PROGRAM Circuito_L12
VAR_INPUT
	Modo_Calibrar_L12: BOOL;
END_VAR
VAR
	fbBomba_L12 :Equipo_Motor_ATV320;
	ControlValv_ioLink_V1:ControlValv_ioLink;
	ControlValv_ioLink_V2: ControlValv_ioLink;
	ControlValv_ioLink_V3: ControlValv_ioLink;
	ControlValv_ioLink_V4: ControlValv_ioLink;
	Falla_L12_V1:BOOL;
	Falla_L12_V2:BOOL;
	Falla_L12_V3:BOOL;
	Falla_L12_V4:BOOL;
	Balanza_PU3_WT12: Balanza;
	dHS:DINT;
	TOF_calibradoIBC: TOF;
	PID_L12_SP:REAL;
	PID_L12_auto:BOOL;
	PID_L12_reset:BOOL;
	PID_L12_manual:REAL;
	PID_L12_bMuerta:REAL := 5;
	PID_L12_Kp:REAL := 0.1;
	PID_L12_Ti:REAL := 100;
	PID_L12_PV:REAL;
	Dosis_L12:REAL;
	TiempoInyeccion_L12	:DINT;
	Peso	:REAL;
	Offset_L12:REAL;
	Inyeccion_L12:BOOL;

	Volumen_L12:REAL;
	Calculo_caudal_L12: Calculo_caudal;
	CorrecionCaudalxOffset_L12: CorrecionCaudalxOffset;
	tInyeccion: TON;
	Total :REAL;
	Totalant	:REAL;
	auxIniCal:BOOL;
	AuxVol12:REAL;
	TDemoraInyectar: TON;
	SetDemoraInyeccion: REAL;
	Tiempo_seg_to_TIME_DemoraInyec: Tiempo_seg_to_TIME;
	AuxTDemoraInyec: TIME;
	PID_L12: FB_PID;
	Tiempo_TIME_to_seg_InyCal: Tiempo_TIME_to_seg;
	AuxInyCal:TIME;
	IniTotalFT2:REAL;
	Auxconsumo:REAL;
	ProductoAsociado: STRING;
	Lavagem_Circuito12: Lavagem;
	Filtro:Filtro2;
	BasicPID_L12: FB_BasicPID;
	TON_StartBomba: TON;
END_VAR

VAR PERSISTENT
	UltimaCalibracao	:UDINT;	//Data e hora da ultima calibração
END_VAR
VAR // added by the converter: edge detectors and wires of the graphical bodies
    _w1, _w2, _w3, _w4, _w5, _w6, _w7, _w8, _w9, _w10, _w11, _w12, _w13 : BOOL;
    _ft1 : F_TRIG;
    _rt1, _rt2, _rt3 : R_TRIG;
END_VAR

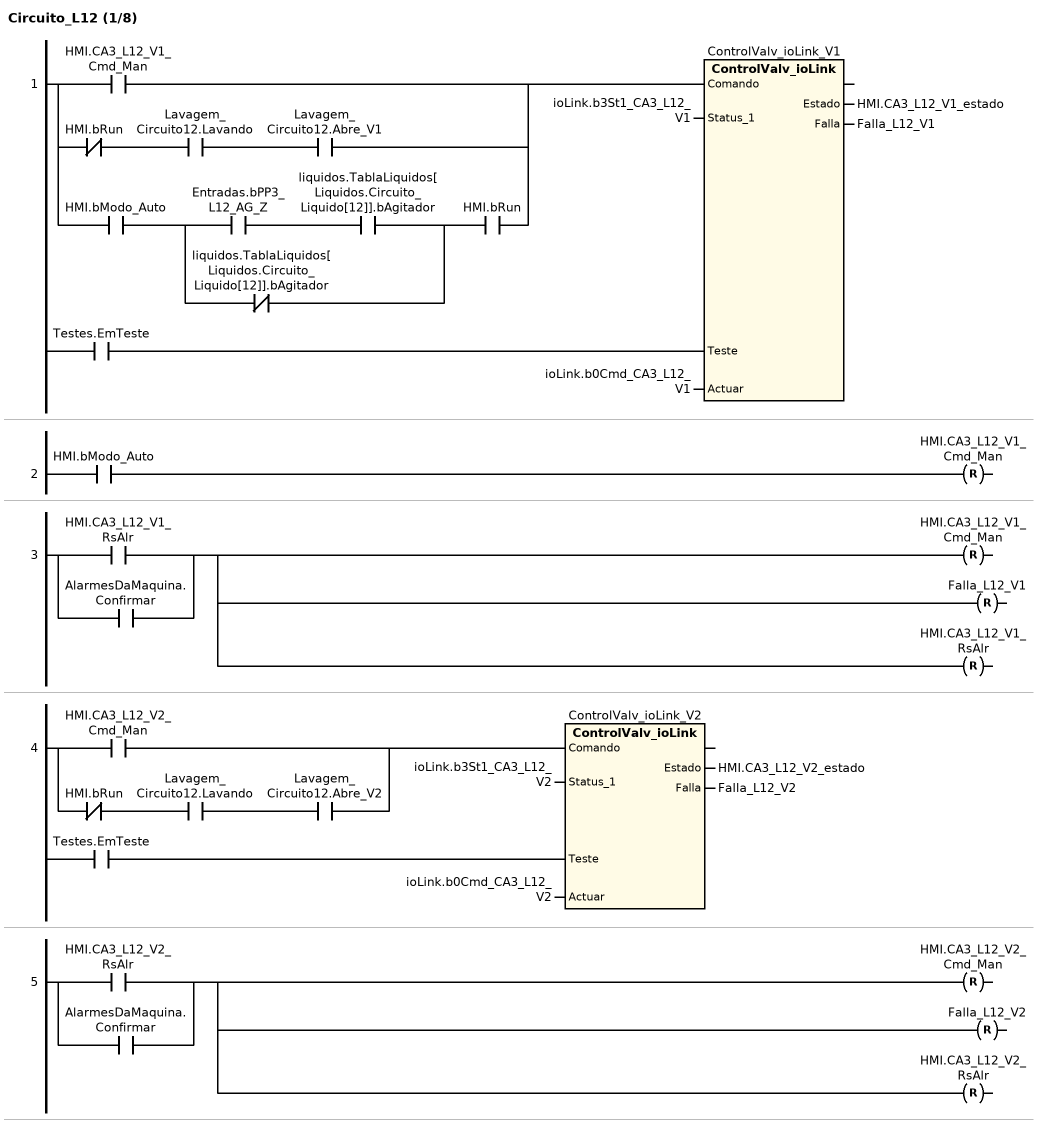
// NETWORK 1
ControlValv_ioLink_V1(
    Comando := HMI.CA3_L12_V1_Cmd_Man OR NOT HMI.bRun AND Lavagem_Circuito12.Lavando AND Lavagem_Circuito12.Abre_V1 OR HMI.bModo_Auto AND (Entradas.bPP3_L12_AG_Z AND (liquidos.TablaLiquidos[Liquidos.Circuito_Liquido[12]].bAgitador) OR NOT (liquidos.TablaLiquidos[Liquidos.Circuito_Liquido[12]].bAgitador)) AND HMI.bRun,
    Status_1 := ioLink.b3St1_CA3_L12_V1,
    Teste := Testes.EmTeste,
    Actuar := ioLink.b0Cmd_CA3_L12_V1,
    Estado => HMI.CA3_L12_V1_estado,
    Falla => Falla_L12_V1); // ControlValv_ioLink

// NETWORK 2
HMI.CA3_L12_V1_Cmd_Man R= HMI.bModo_Auto;

// NETWORK 3
_w1 := HMI.CA3_L12_V1_RsAlr OR AlarmesDaMaquina.Confirmar;
HMI.CA3_L12_V1_Cmd_Man R= _w1;
Falla_L12_V1 R= _w1;
HMI.CA3_L12_V1_RsAlr R= _w1;

// NETWORK 4
ControlValv_ioLink_V2(
    Comando := HMI.CA3_L12_V2_Cmd_Man OR NOT HMI.bRun AND Lavagem_Circuito12.Lavando AND Lavagem_Circuito12.Abre_V2,
    Status_1 := ioLink.b3St1_CA3_L12_V2,
    Teste := Testes.EmTeste,
    Actuar := ioLink.b0Cmd_CA3_L12_V2,
    Estado => HMI.CA3_L12_V2_estado,
    Falla => Falla_L12_V2); // ControlValv_ioLink

// NETWORK 5
_w2 := HMI.CA3_L12_V2_RsAlr OR AlarmesDaMaquina.Confirmar;
HMI.CA3_L12_V2_Cmd_Man R= _w2;
Falla_L12_V2 R= _w2;
HMI.CA3_L12_V2_RsAlr R= _w2;

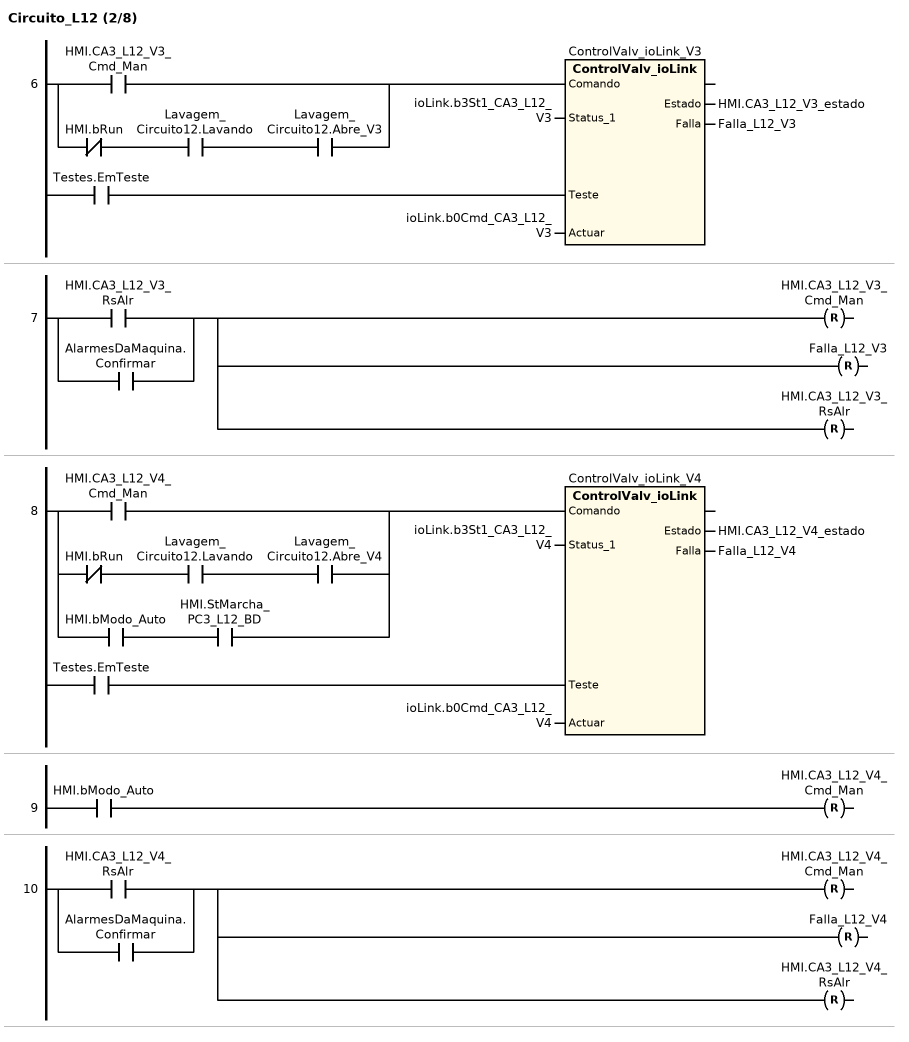
// NETWORK 6
ControlValv_ioLink_V3(
    Comando := HMI.CA3_L12_V3_Cmd_Man OR NOT HMI.bRun AND Lavagem_Circuito12.Lavando AND Lavagem_Circuito12.Abre_V3,
    Status_1 := ioLink.b3St1_CA3_L12_V3,
    Teste := Testes.EmTeste,
    Actuar := ioLink.b0Cmd_CA3_L12_V3,
    Estado => HMI.CA3_L12_V3_estado,
    Falla => Falla_L12_V3); // ControlValv_ioLink

// NETWORK 7
_w3 := HMI.CA3_L12_V3_RsAlr OR AlarmesDaMaquina.Confirmar;
HMI.CA3_L12_V3_Cmd_Man R= _w3;
Falla_L12_V3 R= _w3;
HMI.CA3_L12_V3_RsAlr R= _w3;

// NETWORK 8
ControlValv_ioLink_V4(
    Comando := HMI.CA3_L12_V4_Cmd_Man OR NOT HMI.bRun AND Lavagem_Circuito12.Lavando AND Lavagem_Circuito12.Abre_V4 OR HMI.bModo_Auto AND HMI.StMarcha_PC3_L12_BD,
    Status_1 := ioLink.b3St1_CA3_L12_V4,
    Teste := Testes.EmTeste,
    Actuar := ioLink.b0Cmd_CA3_L12_V4,
    Estado => HMI.CA3_L12_V4_estado,
    Falla => Falla_L12_V4); // ControlValv_ioLink

// NETWORK 9
HMI.CA3_L12_V4_Cmd_Man R= HMI.bModo_Auto;

// NETWORK 10
_w4 := HMI.CA3_L12_V4_RsAlr OR AlarmesDaMaquina.Confirmar;
HMI.CA3_L12_V4_Cmd_Man R= _w4;
Falla_L12_V4 R= _w4;
HMI.CA3_L12_V4_RsAlr R= _w4;

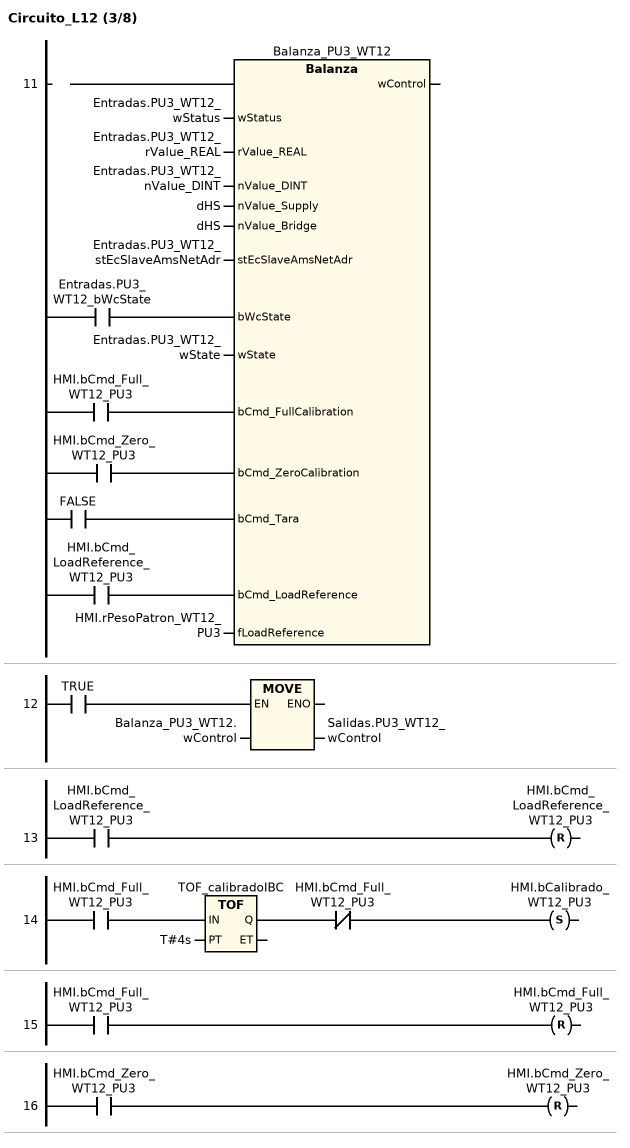
// NETWORK 11
Balanza_PU3_WT12(
    wStatus := Entradas.PU3_WT12_wStatus,
    rValue_REAL := Entradas.PU3_WT12_rValue_REAL,
    nValue_DINT := Entradas.PU3_WT12_nValue_DINT,
    nValue_Supply := dHS,
    nValue_Bridge := dHS,
    stEcSlaveAmsNetAdr := Entradas.PU3_WT12_stEcSlaveAmsNetAdr,
    bWcState := Entradas.PU3_WT12_bWcState,
    wState := Entradas.PU3_WT12_wState,
    bCmd_FullCalibration := HMI.bCmd_Full_WT12_PU3,
    bCmd_ZeroCalibration := HMI.bCmd_Zero_WT12_PU3,
    bCmd_Tara := FALSE,
    bCmd_LoadReference := HMI.bCmd_LoadReference_WT12_PU3,
    fLoadReference := HMI.rPesoPatron_WT12_PU3); // Balanza

// NETWORK 12
Salidas.PU3_WT12_wControl := Balanza_PU3_WT12.wControl;

// NETWORK 13
HMI.bCmd_LoadReference_WT12_PU3 R= HMI.bCmd_LoadReference_WT12_PU3;

// NETWORK 14
TOF_calibradoIBC(IN := HMI.bCmd_Full_WT12_PU3, PT := T#4s); // TOF
HMI.bCalibrado_WT12_PU3 S= TOF_calibradoIBC.Q AND NOT HMI.bCmd_Full_WT12_PU3;

// NETWORK 15
HMI.bCmd_Full_WT12_PU3 R= HMI.bCmd_Full_WT12_PU3;

// NETWORK 16
HMI.bCmd_Zero_WT12_PU3 R= HMI.bCmd_Zero_WT12_PU3;

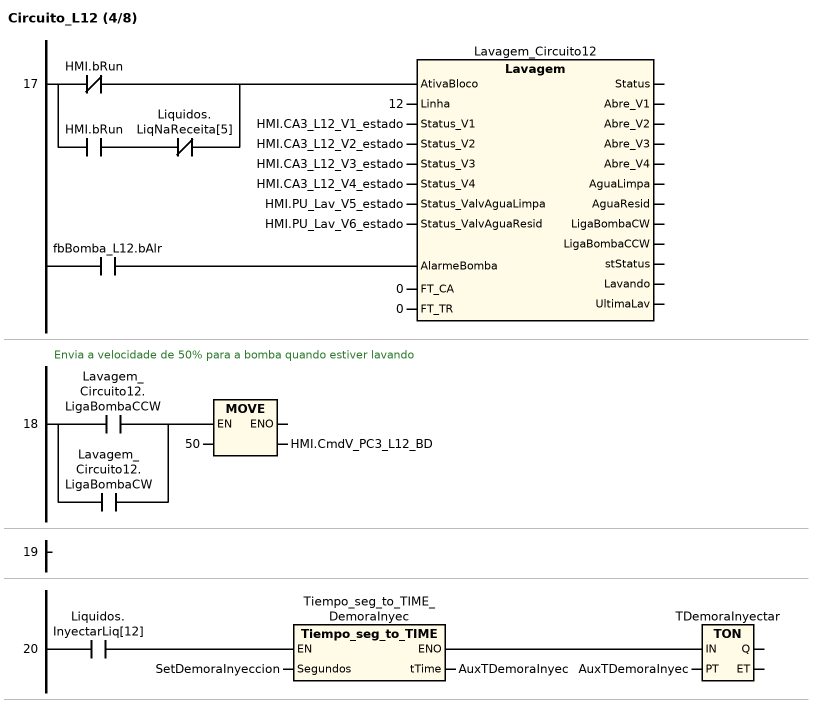
// NETWORK 17
Lavagem_Circuito12(
    AtivaBloco := NOT HMI.bRun OR HMI.bRun AND NOT Liquidos.LiqNaReceita[5],
    Linha := 12,
    Status_V1 := HMI.CA3_L12_V1_estado,
    Status_V2 := HMI.CA3_L12_V2_estado,
    Status_V3 := HMI.CA3_L12_V3_estado,
    Status_V4 := HMI.CA3_L12_V4_estado,
    Status_ValvAguaLimpa := HMI.PU_Lav_V5_estado,
    Status_ValvAguaResid := HMI.PU_Lav_V6_estado,
    AlarmeBomba := fbBomba_L12.bAlr,
    FT_CA := 0,
    FT_TR := 0); // Lavagem

// NETWORK 18
// Envia a velocidade de 50% para a bomba quando estiver lavando
IF Lavagem_Circuito12.LigaBombaCCW OR Lavagem_Circuito12.LigaBombaCW THEN HMI.CmdV_PC3_L12_BD := 50; END_IF

// NETWORK 19

// NETWORK 20
_w5 := Liquidos.InyectarLiq[12];
IF _w5 THEN
    Tiempo_seg_to_TIME_DemoraInyec(Segundos := SetDemoraInyeccion, tTime => AuxTDemoraInyec); // Tiempo_seg_to_TIME
END_IF
TDemoraInyectar(IN := _w5, PT := AuxTDemoraInyec); // TON

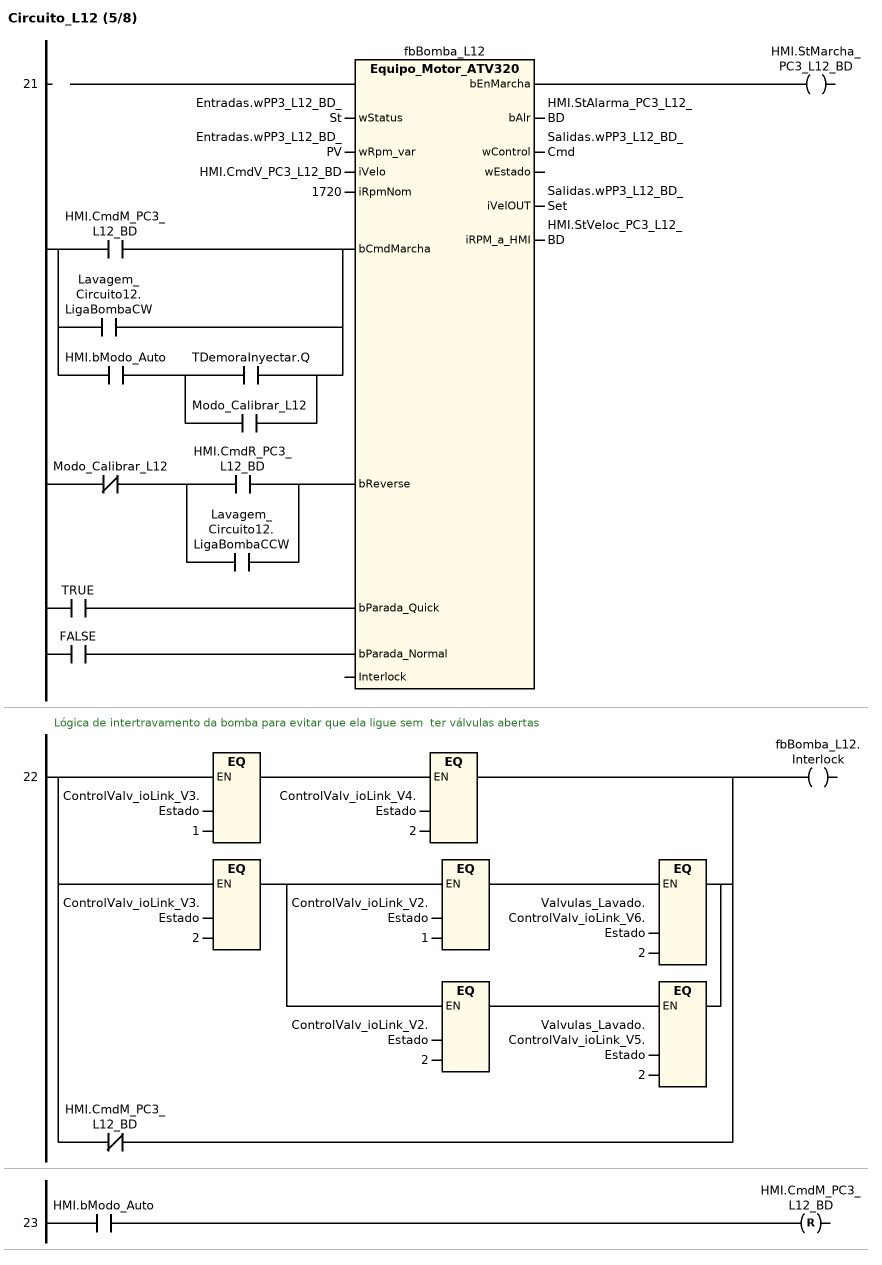
// NETWORK 21
fbBomba_L12(
    wStatus := Entradas.wPP3_L12_BD_St,
    wRpm_var := Entradas.wPP3_L12_BD_PV,
    iVelo := HMI.CmdV_PC3_L12_BD,
    iRpmNom := 1720,
    bCmdMarcha := HMI.CmdM_PC3_L12_BD OR Lavagem_Circuito12.LigaBombaCW OR HMI.bModo_Auto AND (TDemoraInyectar.Q OR Modo_Calibrar_L12),
    bReverse := NOT Modo_Calibrar_L12 AND (HMI.CmdR_PC3_L12_BD OR Lavagem_Circuito12.LigaBombaCCW),
    bParada_Quick := TRUE,
    bParada_Normal := FALSE,
    bAlr => HMI.StAlarma_PC3_L12_BD,
    wControl => Salidas.wPP3_L12_BD_Cmd,
    iVelOUT => Salidas.wPP3_L12_BD_Set,
    iRPM_a_HMI => HMI.StVeloc_PC3_L12_BD); // Equipo_Motor_ATV320
HMI.StMarcha_PC3_L12_BD := fbBomba_L12.bEnMarcha;

// NETWORK 22
// Lógica de intertravamento da bomba para evitar que ela ligue sem  ter válvulas abertas
_w6 := NOT HMI.CmdM_PC3_L12_BD;
IF NOT _w6 THEN
    _w7 := ControlValv_ioLink_V3.Estado = 2;
    _w6 := ControlValv_ioLink_V3.Estado = 1 AND ControlValv_ioLink_V4.Estado = 2 OR (_w7 AND ControlValv_ioLink_V2.Estado = 1 AND Valvulas_Lavado.ControlValv_ioLink_V6.Estado = 2 OR _w7 AND ControlValv_ioLink_V2.Estado = 2 AND Valvulas_Lavado.ControlValv_ioLink_V5.Estado = 2);
END_IF
fbBomba_L12.Interlock := _w6;

// NETWORK 23
HMI.CmdM_PC3_L12_BD R= HMI.bModo_Auto;

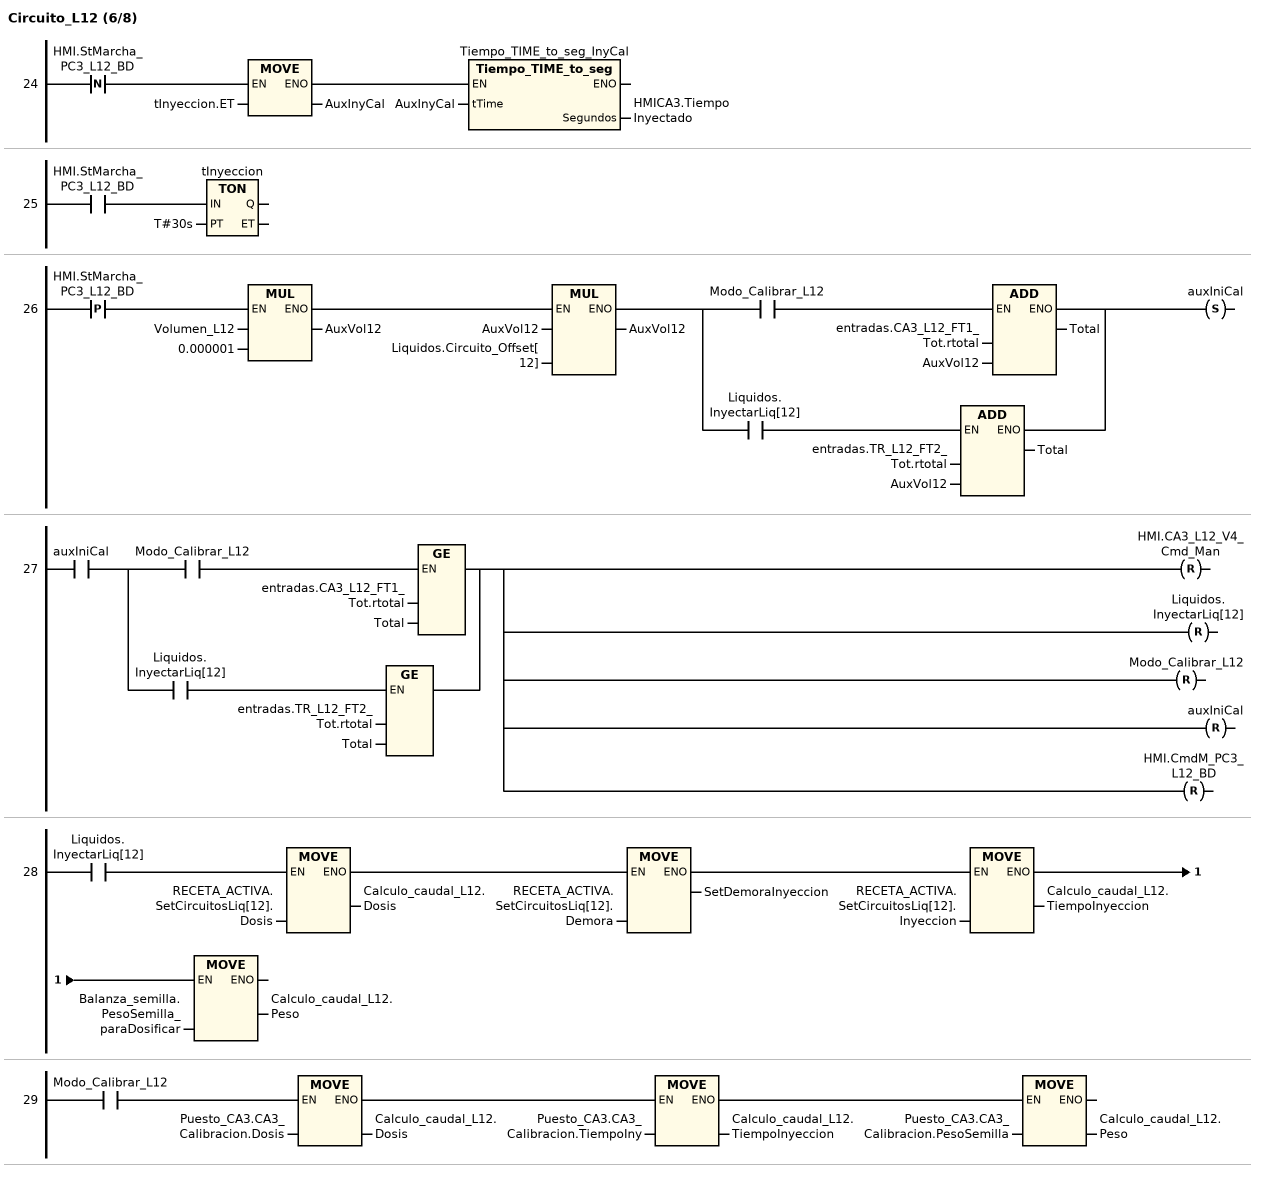
// NETWORK 24
_ft1(CLK := HMI.StMarcha_PC3_L12_BD);
_w8 := _ft1.Q;
IF _w8 THEN AuxInyCal := tInyeccion.ET; END_IF
IF _w8 THEN
    Tiempo_TIME_to_seg_InyCal(tTime := AuxInyCal, Segundos => HMICA3.TiempoInyectado); // Tiempo_TIME_to_seg
END_IF

// NETWORK 25
tInyeccion(IN := HMI.StMarcha_PC3_L12_BD, PT := T#30s); // TON

// NETWORK 26
_rt1(CLK := HMI.StMarcha_PC3_L12_BD);
_w9 := _rt1.Q;
IF _w9 THEN AuxVol12 := Volumen_L12 * 0.000001; END_IF
IF _w9 THEN AuxVol12 := AuxVol12 * Liquidos.Circuito_Offset[12]; END_IF
IF _w9 AND Modo_Calibrar_L12 THEN Total := entradas.CA3_L12_FT1_Tot.rtotal + AuxVol12; END_IF
IF _w9 AND Liquidos.InyectarLiq[12] THEN Total := entradas.TR_L12_FT2_Tot.rtotal + AuxVol12; END_IF
auxIniCal S= _w9 AND Modo_Calibrar_L12 OR _w9 AND Liquidos.InyectarLiq[12];

// NETWORK 27
_w10 := auxIniCal AND Modo_Calibrar_L12 AND entradas.CA3_L12_FT1_Tot.rtotal >= Total OR auxIniCal AND Liquidos.InyectarLiq[12] AND entradas.TR_L12_FT2_Tot.rtotal >= Total;
HMI.CA3_L12_V4_Cmd_Man R= _w10;
Liquidos.InyectarLiq[12] R= _w10;
Modo_Calibrar_L12 R= _w10;
auxIniCal R= _w10;
HMI.CmdM_PC3_L12_BD R= _w10;

// NETWORK 28
_w11 := Liquidos.InyectarLiq[12];
IF _w11 THEN Calculo_caudal_L12.Dosis := RECETA_ACTIVA.SetCircuitosLiq[12].Dosis; END_IF
IF _w11 THEN SetDemoraInyeccion := RECETA_ACTIVA.SetCircuitosLiq[12].Demora; END_IF
IF _w11 THEN Calculo_caudal_L12.TiempoInyeccion := RECETA_ACTIVA.SetCircuitosLiq[12].Inyeccion; END_IF
IF _w11 THEN Calculo_caudal_L12.Peso := Balanza_semilla.PesoSemilla_paraDosificar; END_IF

// NETWORK 29
_w12 := Modo_Calibrar_L12;
IF _w12 THEN Calculo_caudal_L12.Dosis := Puesto_CA3.CA3_Calibracion.Dosis; END_IF
IF _w12 THEN Calculo_caudal_L12.TiempoInyeccion := Puesto_CA3.CA3_Calibracion.TiempoIny; END_IF
IF _w12 THEN Calculo_caudal_L12.Peso := Puesto_CA3.CA3_Calibracion.PesoSemilla; END_IF

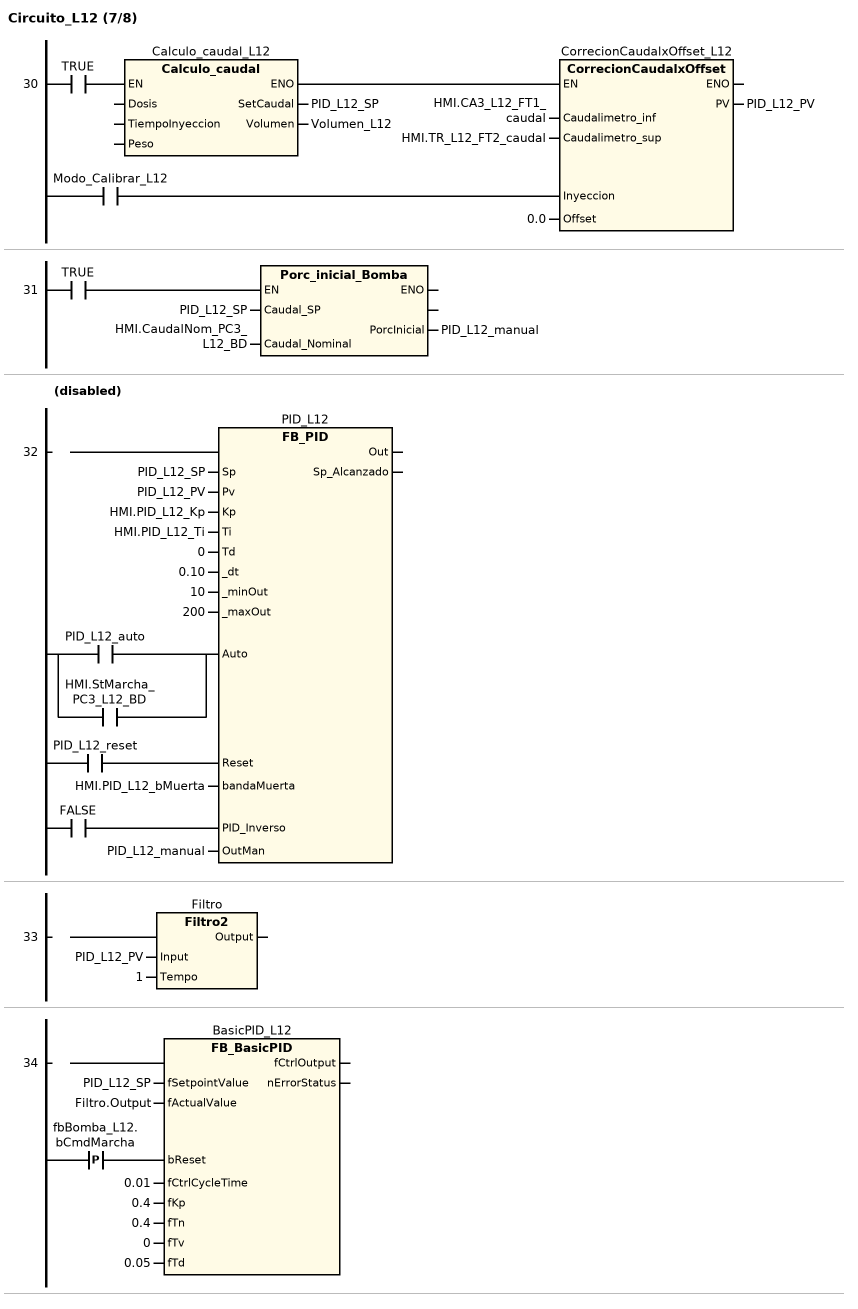
// NETWORK 30
Calculo_caudal_L12(SetCaudal => PID_L12_SP, Volumen => Volumen_L12); // Calculo_caudal
CorrecionCaudalxOffset_L12(
    Caudalimetro_inf := HMI.CA3_L12_FT1_caudal,
    Caudalimetro_sup := HMI.TR_L12_FT2_caudal,
    Inyeccion := Modo_Calibrar_L12,
    Offset := 0.0,
    PV => PID_L12_PV); // CorrecionCaudalxOffset

// NETWORK 31
Porc_inicial_Bomba(Caudal_SP := PID_L12_SP, Caudal_Nominal := HMI.CaudalNom_PC3_L12_BD, PorcInicial => PID_L12_manual);

// NETWORK 32 (disabled)
// PID_L12(
//     Sp := PID_L12_SP,
//     Pv := PID_L12_PV,
//     Kp := HMI.PID_L12_Kp,
//     Ti := HMI.PID_L12_Ti,
//     Td := 0,
//     _dt := 0.10,
//     _minOut := 10,
//     _maxOut := 200,
//     Auto := PID_L12_auto OR HMI.StMarcha_PC3_L12_BD,
//     Reset := PID_L12_reset,
//     bandaMuerta := HMI.PID_L12_bMuerta,
//     PID_Inverso := FALSE,
//     OutMan := PID_L12_manual); // FB_PID

// NETWORK 33
Filtro(Input := PID_L12_PV, Tempo := 1); // Filtro2

// NETWORK 34
_rt2(CLK := fbBomba_L12.bCmdMarcha);
BasicPID_L12(
    fSetpointValue := PID_L12_SP,
    fActualValue := Filtro.Output,
    bReset := _rt2.Q,
    fCtrlCycleTime := 0.01,
    fKp := 0.4,
    fTn := 0.4,
    fTv := 0,
    fTd := 0.05); // FB_BasicPID

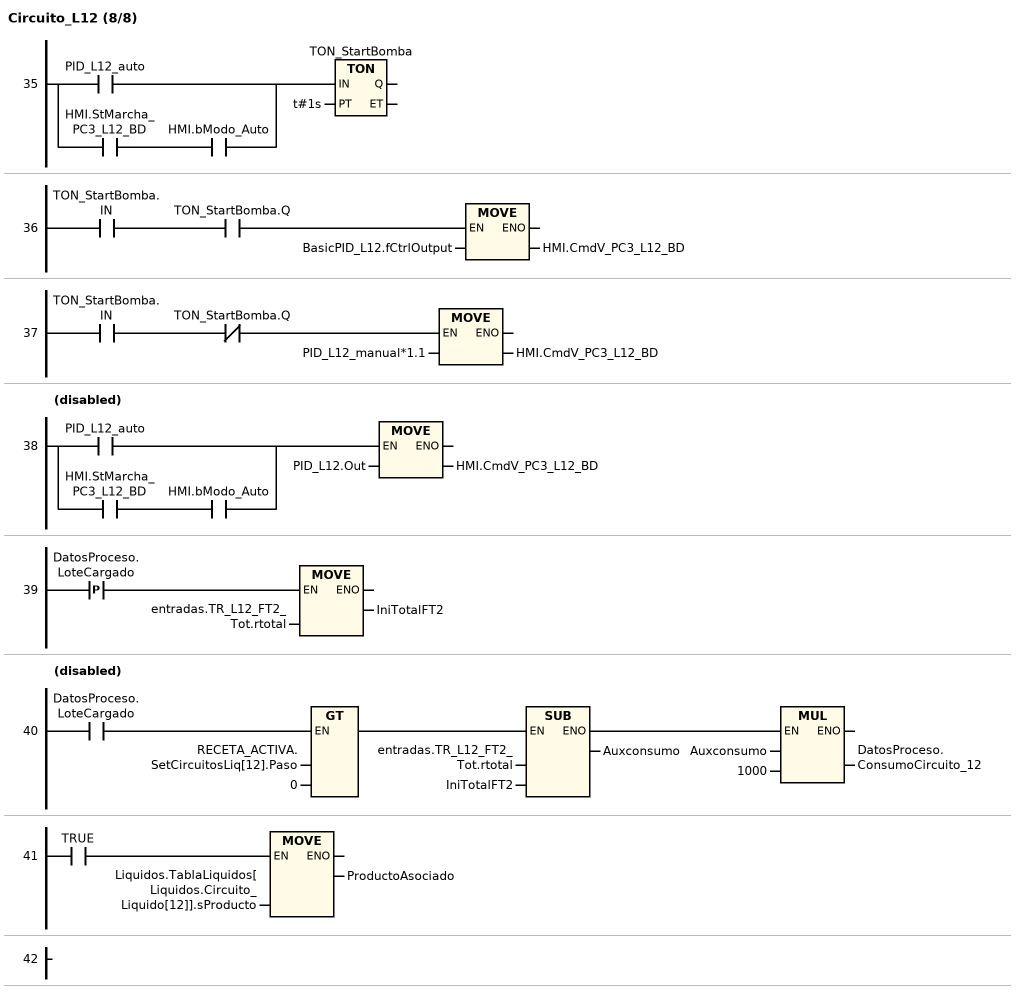
// NETWORK 35
TON_StartBomba(IN := PID_L12_auto OR HMI.StMarcha_PC3_L12_BD AND HMI.bModo_Auto, PT := t#1s); // TON

// NETWORK 36
IF TON_StartBomba.IN AND TON_StartBomba.Q THEN HMI.CmdV_PC3_L12_BD := BasicPID_L12.fCtrlOutput; END_IF

// NETWORK 37
IF TON_StartBomba.IN AND NOT TON_StartBomba.Q THEN HMI.CmdV_PC3_L12_BD := PID_L12_manual*1.1; END_IF

// NETWORK 38 (disabled)
// IF PID_L12_auto OR HMI.StMarcha_PC3_L12_BD AND HMI.bModo_Auto THEN HMI.CmdV_PC3_L12_BD := PID_L12.Out; END_IF

// NETWORK 39
_rt3(CLK := DatosProceso.LoteCargado);
IF _rt3.Q THEN IniTotalFT2 := entradas.TR_L12_FT2_Tot.rtotal; END_IF

// NETWORK 40 (disabled)
// _w13 := DatosProceso.LoteCargado AND RECETA_ACTIVA.SetCircuitosLiq[12].Paso > 0;
// IF _w13 THEN Auxconsumo := entradas.TR_L12_FT2_Tot.rtotal - IniTotalFT2; END_IF
// IF _w13 THEN DatosProceso.ConsumoCircuito_12 := Auxconsumo * 1000; END_IF

// NETWORK 41
ProductoAsociado := Liquidos.TablaLiquidos[Liquidos.Circuito_Liquido[12]].sProducto;

// NETWORK 42

END_PROGRAM

(* stored: Version 1.1.0.1, ProductVersion 3.1.4024.14
   POU Circuito_L12: Id {53874b89-bd1f-478e-943e-5aaaa9701307}, SpecialFunc None *)
